Staubli VAL3: start.pgx

program start()
  local num l_nBin[3]
  local num l_nRes
  local num l_nRows
  local num l_nCols
  local num l_nCounter
  local num l_nIndices[2]
  local string l_sString[10]
begin

  ? "## test num2Bool"
  ? "nTest[0] = nTest[1] = nTest[4] = 1"
  nTest[0] = nTest[1] = nTest[4] = 1

  call num2bool(nTest, bResult, bError)
  call printBool(bResult)

  ? "## test countBool"
  call countBool(bResult,nResult)
  call printNum(nResult)

  ? "## test allBool"
  call allBool(bResult, bResult2)
  call printBool(bResult2)

  ? "## test allBool"
  ? "nTest[2] = nTest[3] = 1"
  nTest[2] = nTest[3] = 1
  call num2bool(nTest, bResult, bError)
  call allBool(bResult, bResult2)
  call printBool(bResult2)

  ? "## test countBool"
  call countBool(bResult,nResult)
  call printNum(nResult)

  ? "## test anyBool TRUE"
  call anyBool(bResult, "TRUE",bResult2)
  call printBool(bResult2)

  ? "## test anyBool FALSE"
  call anyBool(bResult, "FALSE",bResult2)
  call printBool(bResult2)

  ? "## test bool2num"
  call bool2num(bResult, nResult, bError)
  call printNum(nResult)

  ? "## test bool2num"
  ? "nTest[0] = nTest[1] = nTest[4] = 0"
  nTest[0] = nTest[1] = nTest[4] = 0
  call num2bool(nTest, bResult, bError)
  call bool2num(bResult, nResult, bError)
  call printNum(nResult)

  ? "## test bin2dec"
  ? "nTest"
  l_nBin[0] = 1
  l_nBin[1] = 0
  l_nBin[2] = 0

  call bin2dec(l_nBin, l_nRes)
  call printNum(l_nRes)

  ? "## test mergeVectors"
  nTest2[0] = 5
  nTest2[1] = -3
  nTest2[2] = 10
  nTest2[4] = -1

  call mergeVectors(nTest, nTest2, nResult)
  call printNum(nResult)

  ? "## test colSum"
  for l_nRows = 0 to size(nMatrix,1)-1
    for l_nCols = 0 to size(nMatrix,2)-1
      nMatrix[l_nRows,l_nCols] = l_nCounter
      l_nCounter = l_nCounter +1
    endFor
  endFor

  // 0 1  2  3
  // 4 5  6  7
  // 8 9 10 11

  ? "## Matrix to analyse:"
  call printNum2d(nMatrix)

  call colSum(nMatrix, nResult)
  call printNum(nResult)

  ? "## test rowSum"
  call rowSum(nMatrix, nResult)
  call printNum(nResult)

  ? "## test extractRow"
  call extractRow(nMatrix, 2, nResult)
  call printNum(nResult)

  ? "## test extractRows"
  l_nIndices[0] = 2
  l_nIndices[1] = 1
  call extractRows(nMatrix, l_nIndices, nResult2D)
  call printNum2d(nResult2D)

  ? "## test extractCol"
  call extractCol(nMatrix, 3, nResult)
  call printNum(nResult)

  ? "## test extractGrid: rows"
  call extractGrid(nMatrix, 1, 2,0,nResult2D)
  call printNum2d(nResult2D)

  ? "## test extractGrid: cols"
  call extractGrid(nMatrix, 2, 3,0,nResult2D)
  call printNum2d(nResult2D)

  ? "## test repeat(nTest2,3)"
  call repeat(nTest2,3, nResult)
  call printNum(nResult)

  ? "## test uniqueStr()"
  l_sString[0] = "A"
  l_sString[1] = "B"
  l_sString[2] = "C"
  l_sString[3] = "A"
  l_sString[4] = "B"
  l_sString[5] = "B"
  l_sString[6] = "a"
  l_sString[7] = "D"
  l_sString[8] = "V"
  l_sString[9] = "G"

  call uniqueStr(l_sString, sResult)
  call printStr(sResult)


end
